// TIA Portal project "VGR_demo_rev2.0" (V16)

(* hardware
DEVICE "S7-1200 station_1"  S7-1200 Station
   slot 0: "Rack_0"  S7-1200 Rack  Rack  V1.0
   slot 1: "PLC_1"  CPU 1214C DC/DC/DC  6ES7 214-1AG40-0XB0  V4.4
   slot 2: "DI 16x24VDC/DQ 16xRelay_1"  6ES7 223-1BL32-0XB0  V2.0
   slot 3: "DI 16x24VDC/DQ 16xRelay_2"  6ES7 223-1BL32-0XB0  V2.0
*)

// ===== PLC "PLC_1"  CPU 1214C DC/DC/DC =====

VAR_GLOBAL   // PLC tag table "VGR - Vacuum Gripper Robot"
   "IX_VGR_RefSwitchVerticalAxis_I1" AT %I12.0 : Bool;   // VGR - I1 = Reference switch vertical axis
   "IX_VGR_RefSwitchHorizontalAxis_I2" AT %I12.1 : Bool;   // VGR - I2 = Reference switch horizontal axis
   "IX_VGR_RefSwitchRotate_I3" AT %I12.2 : Bool;   // VGR - I3 = Reference switch rotate
   "QX_VGR_M1_VerticalAxisUp_Q1" AT %Q13.0 : Bool;   // VGR - Q1 = Motor M1 vertical axis up
   "QX_VGR_M1_VerticalAxisDown_Q2" AT %Q13.1 : Bool;   // VGR - Q2 = Motor M1 vertical axis down
   "QX_VGR_M2_HorizontalAxisBackward_Q3" AT %Q13.2 : Bool;   // VGR - Q3 = Motor M2 horizontal axis backward
   "QX_VGR_M2_HorizontalAxisForward_Q4" AT %Q13.3 : Bool;   // VGR - Q4 = Motor M2 horizontal axis forward
   "QX_VGR_M3_RotateClockwise_Q5" AT %Q13.4 : Bool;   // VGR - Q5 = Motor M3 rotate clockwise
   "QX_VGR_M3_RotateCounterclockwise_Q6" AT %Q13.5 : Bool;   // VGR - Q6 = Motor M3 rotate counterclockwise
   "QX_VGR_Compressor_Q7" AT %Q13.6 : Bool;   // VGR - Q7 = Compressor
   "QX_VGR_ValveVacuum_Q8" AT %Q13.7 : Bool;   // VGR - Q8 = Valve vacuum
   "Enc_VGR_vertical" AT %ID1008 : DInt;
   "Enc_VGR_horizontal" AT %ID1012 : DInt;
   "Enc_VGR_rotate" AT %ID1016 : DInt;
END_VAR

VAR_GLOBAL   // PLC tag table "MPO - Multi Processing Station with Oven"
   "IX_MPO_RefSwitchOvenFeederInside_I6" AT %I8.5 : Bool;   // MPO - I6 = Reference switch oven feeder inside
   "IX_MPO_RefSwitchOvenFeederOutside_I7" AT %I8.6 : Bool;   // MPO - I7 = Reference switch oven feeder outside
   "QX_MPO_M4_OvenFeederRetract_Q5" AT %Q8.2 : Bool;   // MPO - Q5 = Motor M4 oven feeder retract
   "QX_MPO_M4_OvenFeederExtend_Q6" AT %Q8.3 : Bool;   // MPO - Q6 = Motor M4 oven feeder extend
   "QX_MPO_Compressor_Q10" AT %Q8.7 : Bool;   // MPO - Q10 = Compressor
   "QX_MPO_ValveOvenDoor_Q13" AT %Q9.2 : Bool;   // MPO - Q13 = Valve oven door
END_VAR

TYPE "typ_History"
   STRUCT
      ldt_ts : DTL;
      i_code : Int;
   END_STRUCT;
END_TYPE

TYPE "typ_Workpiece"
   STRUCT
      s_id : String;
      s_type : String;
      s_state : String;
   END_STRUCT;
END_TYPE

TYPE "typ_VGR"
   STRUCT
      x_Start_Park_Position : Bool;
      x_Park_Position_Reached : Bool;
      x_NFC_Start_First : Bool;
      x_NFC_Start : Bool;
      x_NFC_Completed : Bool;
      x_HBW_Storage : Bool;
      x_HBW_Outsource : Bool;
      s_HBW_Outsource_Typ : String;
      x_HBW_Discards : Bool;
      x_HBW_PickedUp : Bool;
      x_MPO_Req_Discard : Bool;
      x_MPO_Discards : Bool;
      x_Ready_For_Outsource : Bool;
      x_State_Process : Bool;
      x_Workpiece_NiO : Bool;
      horizontal_Axis : "typ_Axis";
      vertical_Axis : "typ_Axis";
      rotate_Axis : "typ_Axis";
      Workpiece : "typ_Workpiece";
      History : Array[1..20] of "typ_History";
      di_Pos_DSI_horizontal : DInt;
      di_Pos_DSI_Collect_vertical : DInt;
      di_Pos_DSI_Discard_vertical : DInt;
      di_Offset_Pos_DSI_NFC_vertical : DInt;
      di_Pos_DSI_rotate : DInt;
      di_Pos_DSO_horizontal : DInt;
      di_Pos_DSO_Collect_vertical : DInt;
      di_Pos_DSO_Discard_vertical : DInt;
      di_Offset_Pos_DSO_vertical : DInt;
      di_Pos_DSO_rotate : DInt;
      di_Pos_Color_horizontal : DInt;
      di_Pos_Color_vertical : DInt;
      di_Pos_Color_rotate : DInt;
      di_Pos_NFC_horizontal : DInt;
      di_Pos_NFC_vertical : DInt;
      di_Pos_NFC_rotate : DInt;
      di_Pos_MPO_horizontal : DInt;
      di_Pos_MPO_vertical : DInt;
      di_Offset_Pos_MPO_vertical : DInt;
      di_Pos_MPO_rotate : DInt;
      di_Pos_HBW_horizontal : DInt;
      di_Offset_Pos_HBW_horizontal : DInt;
      di_Pos_HBW_Collect_vertical : DInt;
      di_Pos_HBW_Discard_vertical : DInt;
      di_Offset_Pos_HBW_vertical : DInt;
      di_Pos_HBW_rotate : DInt;
      di_Pos_NiO_horizontal : DInt;
      di_Pos_NiO_vertical : DInt;
      di_Pos_NiO_rotate : DInt;
      di_Pos_SLD_Blue_horizontal : DInt;
      di_Pos_SLD_Blue_vertical : DInt;
      di_Pos_SLD_Blue_rotate : DInt;
      di_Pos_SLD_Red_horizontal : DInt;
      di_Pos_SLD_Red_vertical : DInt;
      di_Pos_SLD_Red_rotate : DInt;
      di_Pos_SLD_White_horizontal : DInt;
      di_Pos_SLD_White_vertical : DInt;
      di_Pos_SLD_White_rotate : DInt;
      di_Pos_Park_horizontal : DInt;
      di_Pos_Park_vertical : DInt;
      di_Pos_Park_rotate : DInt;
   END_STRUCT;
END_TYPE

TYPE "typ_SetupAxis"
   STRUCT
      x_Setup_Activ : Bool;   // Einrichten Kalibrieren aktiv / Set up calibration active
      i_AxisSelection : Int;   // Nummer der Achse / Number of the axis
      i_Function : Int;   // 0= Automatic, 10=Ref. Fahrt, 20= Tippen, 30=Tippen mit Schritweite, 40= Pos. Anfahren / 0 = automatic, 10 = ref. Travel, 20 = tap, 30 = tap with step width, 40 = start
      x_Set_Ref_Pos : Bool;   // Referenzwert setzen / Set reference value
      x_Set_Soft_End_Pos : Bool;   // Softwareendlagen setzen / Set software end positions
      x_Approach_Ref_Pos : Bool;   // Referenz anfahren / Approach reference
      x_Axis_Pos : Bool;   // Achse positiv / Axis positiv
      x_Axis_Neg : Bool;   // Achse negativ / Axis negative
      x_Approach_Target_Pos : Bool;   // Zielposition anfahren / Approach Target position
      w_Increment : Word;   // Inkremente pro Schritt / Increments per step
      i_PWM : Int;   // PWM Signal
      di_Target_Position : DInt;   // Zielposition / Target position
      di_ActualPosition : DInt;   // Aktuelle Position / Actual position
      di_Ref_Pos : DInt;   // Referenzposition / Reference position
      di_Actual_Ref_Pos : DInt;   // Aktuelle Referenzposition / Current reference position
      di_Soft_End_Pos_Neg : DInt;   // Softwareendlage negativ / Software end position negative
      di_Actual_Soft_End_Pos_Neg : DInt;   // Aktuelle Softwareendlage negativ / Current software end position negative
      di_Soft_End_Pos_Pos : DInt;   // Softwareendlage positiv / Software end position positiv
      di_Actual_Soft_End_Pos_Pos : DInt;   // Aktuelle Softwareendlage positiv / Current software end position positiv
      di_LoopValue : DInt;   // Schleifenwert / Loop value
   END_STRUCT;
END_TYPE

TYPE "typ_Axis_Data"
   STRUCT
      di_Pos_Soft_Switch : DInt := 0;
      di_Neg_Soft_Switch : DInt := 0;
      di_Ref_Pos : DInt := 0;
      di_Loop_Value : DInt := 0;
      di_Pos_Window : DInt := 15;
   END_STRUCT;
END_TYPE

TYPE "typ_Axis"
   STRUCT
      x_Start_Positioning : Bool;
      x_Reference : Bool;
      x_Referenced : Bool;
      x_Position_Reached : Bool;
      di_Target_Position : DInt;
      di_Increment : DInt;
      di_Actual_Position : DInt := 0;
      i_PWM : Int;
      Config : "typ_Axis_Data";
   END_STRUCT;
END_TYPE

TYPE "typ_Setup"
   STRUCT
      x_Clean_Rack_HBW : Bool;
      x_Park_Position : Bool;
      x_AcknowledgeButton : Bool;
      x_Color_Sensor_Calibration : Bool;
      x_Set_Calib_Value_Color_Blue : Bool;
      x_Set_Calib_Value_Color_White : Bool;
      x_Set_Calib_Value_Color_Red : Bool;
      x_Calculate_Value_Color : Bool;
      i_Color_Sensor_Selection : Int;
      w_Calib_ColorValue_Blue : Word;
      w_Calib_ColorValue_White : Word;
      w_Calib_ColorValue_Red : Word;
      w_Threshold_White_Red : Word;
      w_Threshold_Red_Blue : Word;
      w_Actual_ColorValue : Word;
      x_Set_Pos_Activ : Bool;   // Einrichten Kalibrieren aktiv / Set up calibration active
      x_Start_Positioning : Bool;
      x_Final_Positioning : Bool;
      x_Home_Positioning : Bool;
      x_Start_Offset : Bool;
      i_Pos_Selection : Int;   // Nummer der Achse / Number of the axis
      di_Pos_Horizontal : DInt;
      di_Pos_Vertical : DInt;
      di_Pos_Rotate : DInt;
      x_Counter_Value_Calibration : Bool;   // Einrichten Kalibrieren aktiv
      i_Calib_CounterValue_Blue : Int := 26;
      i_Calib_CounterValue_White : Int := 5;
      i_Calib_CounterValue_Red : Int := 16;
      x_Set_CounterValues : Bool;   // Einrichten Kalibrieren aktiv
      x_Activate_Continuous_Operation : Bool;
   END_STRUCT;
END_TYPE

// folder: 3.1. VGR

DATA_BLOCK "PRG_VGR_Demo_DB"   // DB1
{ S7_Optimized_Access := 'TRUE' }
VERSION : 0.1
// stored: InstanceOfName PRG_VGR_Demo
"PRG_VGR_Demo"
BEGIN
   di_Pos_Second_rotate := 885;
   di_Pos_Second_vertical_high := 450;
END_DATA_BLOCK

DATA_BLOCK "PRG_VGR_Axis_horizontal_DB"   // DB8
{ S7_Optimized_Access := 'TRUE' }
VERSION : 0.1
// stored: InstanceOfName PRG_VGR_Axis_horizontal
"PRG_VGR_Axis_horizontal"
BEGIN
END_DATA_BLOCK

DATA_BLOCK "PRG_VGR_Axis_vertical_DB"   // DB9
{ S7_Optimized_Access := 'TRUE' }
VERSION : 0.1
// stored: InstanceOfName PRG_VGR_Axis_vertical
"PRG_VGR_Axis_vertical"
BEGIN
END_DATA_BLOCK

DATA_BLOCK "PRG_VGR_Axis_rotate_DB"   // DB10
{ S7_Optimized_Access := 'TRUE' }
VERSION : 0.1
// stored: InstanceOfName PRG_VGR_Axis_rotate
"PRG_VGR_Axis_rotate"
BEGIN
END_DATA_BLOCK

DATA_BLOCK "PRG_VGR_Axis_horizontal_Act_Pos_DB"   // DB15
{ S7_Optimized_Access := 'TRUE' }
VERSION : 0.1
// stored: InstanceOfName PRG_VGR_Axis_horizontal_Act_Pos
"PRG_VGR_Axis_horizontal_Act_Pos"
BEGIN
END_DATA_BLOCK

DATA_BLOCK "PRG_VGR_Axis_vertical_Act_Pos_DB"   // DB29
{ S7_Optimized_Access := 'TRUE' }
VERSION : 0.1
// stored: InstanceOfName PRG_VGR_Axis_vertical_Act_Pos
"PRG_VGR_Axis_vertical_Act_Pos"
BEGIN
END_DATA_BLOCK

DATA_BLOCK "PRG_VGR_Axis_rotate_Act_Pos_DB"   // DB31
{ S7_Optimized_Access := 'TRUE' }
VERSION : 0.1
// stored: InstanceOfName PRG_VGR_Axis_rotate_Act_Pos
"PRG_VGR_Axis_rotate_Act_Pos"
BEGIN
END_DATA_BLOCK

// folder: 4. Global Declaration

DATA_BLOCK "gtyp_VGR"   // DB2
TITLE = Global DB VGR
{ S7_Optimized_Access := 'TRUE' }
AUTHOR : A.Schaefer
VERSION : 0.0
BEGIN
   di_Pos_DSI_Collect_vertical := 2950;
   di_Pos_MPO_vertical := 2000;
   di_Pos_HBW_Discard_vertical := 200;
   vertical_Axis.Config.di_Pos_Soft_Switch := 20000;
   horizontal_Axis.Config.di_Pos_Soft_Switch := 20000;
   rotate_Axis.Config.di_Pos_Soft_Switch := 20000;
   di_Pos_DSI_horizontal := 20;
   di_Pos_DSI_rotate := 30;
   di_Pos_Color_horizontal := 150;
   di_Pos_Color_rotate := 430;
   di_Pos_Color_vertical := 2450;
   di_Pos_NFC_vertical := 2450;
   di_Pos_NFC_horizontal := 900;
   di_Pos_NFC_rotate := 700;
   di_Pos_HBW_rotate := 5350;
   di_Offset_Pos_DSI_NFC_vertical := 1200;
   di_Offset_Pos_HBW_vertical := 100;
   di_Pos_HBW_horizontal := 600;
   di_Pos_SLD_Red_rotate := 1460;
   di_Pos_SLD_White_rotate := 1720;
   di_Pos_SLD_Blue_rotate := 1200;
   di_Pos_SLD_Red_vertical := 3100;
   di_Pos_SLD_White_vertical := 3100;
   di_Pos_SLD_Blue_vertical := 3100;
   di_Pos_SLD_Red_horizontal := 1580;
   di_Pos_SLD_White_horizontal := 1370;
   di_Pos_SLD_Blue_horizontal := 2150;
   di_Pos_DSO_rotate := 970;
   di_Pos_MPO_rotate := 3495;
   di_Pos_NiO_rotate := 1100;
   di_Pos_DSO_horizontal := 2070;
   di_Pos_DSO_Discard_vertical := 1480;
   di_Pos_NiO_vertical := 2700;
   di_Pos_MPO_horizontal := 3300;
   di_Pos_HBW_Collect_vertical := 650;
   di_Offset_Pos_MPO_vertical := 650;
   horizontal_Axis.i_PWM := 500;
   vertical_Axis.i_PWM := 800;
   rotate_Axis.i_PWM := 500;
   di_Offset_Pos_DSO_vertical := 500;
   di_Pos_Park_vertical := 3000;
   di_Pos_Park_rotate := 1750;
   di_Pos_Park_horizontal := 150;
   rotate_Axis.Config.di_Pos_Window := 15;
   vertical_Axis.Config.di_Pos_Window := 15;
   horizontal_Axis.Config.di_Pos_Window := 15;
END_DATA_BLOCK

DATA_BLOCK "gtyp_SetupAxis"   // DB4
TITLE = Global DB Setup Axis
{ S7_Optimized_Access := 'TRUE' }
AUTHOR : A.Schaefer
VERSION : 0.0
BEGIN
END_DATA_BLOCK

DATA_BLOCK "gtyp_Setup"   // DB23
TITLE = Global DB Setup
{ S7_Optimized_Access := 'TRUE' }
AUTHOR : A.Schaefer
VERSION : 0.0
BEGIN
END_DATA_BLOCK

// folder: (top level)

ORGANIZATION_BLOCK "Main"   // OB1, SCL, ProgramCycle
TITLE = "Main Program Sweep (Cycle)"
{ S7_Optimized_Access := 'TRUE' }
AUTHOR : A.Schaefer
VERSION : 0.0
BEGIN
   "PRG_VGR_Axis_horizontal_DB"();
   "PRG_VGR_Axis_vertical_DB"();
   "PRG_VGR_Axis_rotate_DB"();
   "PRG_VGR_Demo_DB"();
END_ORGANIZATION_BLOCK

ORGANIZATION_BLOCK "Cyclic interrupt"   // OB30, SCL, CyclicInterrupt
TITLE = Cyclic interrupt
{ S7_Optimized_Access := 'TRUE' }
AUTHOR : A.Schaefer
VERSION : 0.0
   VAR_TEMP
      li_Return_LDT : Int;
   END_VAR
BEGIN
   "PRG_VGR_Axis_horizontal_Act_Pos_DB"();
   "PRG_VGR_Axis_vertical_Act_Pos_DB"();
   "PRG_VGR_Axis_rotate_Act_Pos_DB"();
END_ORGANIZATION_BLOCK

ORGANIZATION_BLOCK "Startup"   // OB100, SCL, Startup
TITLE = "Complete Restart"
{ S7_Optimized_Access := 'TRUE' }
VERSION : 0.1
   VAR_INPUT
      LostRetentive : Bool;   // True if retentive data are lost
      LostRTC : Bool;   // True if date and time are lost
   END_VAR
BEGIN
   "PRG_VGR_Demo_DB".li_StepCase := 0;
END_ORGANIZATION_BLOCK

// folder: 1. FB / FC

FUNCTION_BLOCK "FB_INC_DEC"   // FB9, SCL
TITLE = Funktionblock Increment decodition
{ S7_Optimized_Access := 'TRUE' }
AUTHOR : A.Schaefer
VERSION : 0.0
   VAR_INPUT
      inx_CHa : Bool := false;
      inx_CHb : Bool := false;
      inx_RST : Bool := False;
      ini_Ref_Wert : Int := 0;
   END_VAR
   VAR_OUTPUT
      outx_dir : Bool := false;
      outi_cnt : Int := 0;
   END_VAR
   VAR
      lx_edgea : Bool := False;
      lx_clka : Bool;
      lx_clkb : Bool;
      lx_edgeb : Bool;
      lx_axb : Bool;
      lx_dir : Bool;
      li_cnt : Int;
   END_VAR
BEGIN

   #lx_axb := #inx_CHa XOR #inx_CHb;

   (* create pulses for channel a *)
   #lx_clka := #inx_CHa XOR #lx_edgea;
   #lx_edgea := #inx_CHa;

   #lx_clkb := #inx_CHb XOR #lx_edgeb;
   #lx_edgeb := #inx_CHb;

   (* create pulses for both channels *)
   #lx_clka := #lx_clka OR #lx_clkb;

   (* set the direction output *)
   IF #lx_axb AND #lx_clka THEN
       #lx_dir := TRUE;
   END_IF;
   IF #lx_axb AND #lx_clkb THEN
       #lx_dir := FALSE;
   END_IF;

   (* increment or decrement the counter *)
   IF #lx_clka AND #lx_dir THEN
       #li_cnt := #li_cnt + 1;
   END_IF;
   IF #lx_clka AND NOT #lx_dir THEN
       #li_cnt := #li_cnt - 1;
   END_IF;

   (* reset the counter if rst active *)
   IF #inx_RST THEN
       #li_cnt := #ini_Ref_Wert;
   END_IF;

   #outx_dir := #lx_dir;
   #outi_cnt := #li_cnt;
END_FUNCTION_BLOCK

FUNCTION_BLOCK "FB_Axis"   // FB22, SCL
TITLE = Functionblock Axis
{ S7_Optimized_Access := 'TRUE' }
AUTHOR : A.Schaefer
VERSION : 0.0
   VAR_INPUT
      ini_Axis : Int;
      indi_Increment : DInt;
      inx_Ref_Switch : Bool;
      inx_Start_Positioning : Bool;
      inx_Referencing : Bool;
      ini_PWM : Int;
      indi_Target_Position : DInt;
   END_VAR
   VAR_OUTPUT
      outx_Referenced : Bool;
      outx_Position_Reached : Bool;
      outx_Motor_Pos : Bool;
      outx_Motor_Neg : Bool;
      outi_Motor_PWM : Int;
      outdi_Actual_Position : DInt;
   END_VAR
   VAR_IN_OUT
      inouttyp_Config : "typ_Axis_Data";
      inouttyp_Setup : "typ_SetupAxis";
   END_VAR
   VAR
      li_StepCaseSetup : Int;
      li_StepCase : Int;
      lx_Init : Bool;
      lx_Motor_Neg : Bool;
      lx_Motor_Pos : Bool;
      lx_Start_TON_Wait : Bool;
      li_PWM : Int;
      ldi_ValueStep : DInt;
      ldi_Actual_Position : DInt;
      ldi_Actual_Position_Old : DInt;
      lfb_R_Trig_Setup : R_TRIG;
      lfb_R_Trig_Referencing : R_TRIG;
      lfb_TON_Wait : TON_TIME;
   END_VAR
BEGIN
   IF #lx_Init THEN

       // rising edge set up axis
       #lfb_R_Trig_Setup(CLK := #inouttyp_Setup.x_Setup_Activ);

       //Reload when switching to set up
       IF #lfb_R_Trig_Setup.Q THEN
           #inouttyp_Setup.di_LoopValue               := #inouttyp_Config.di_Loop_Value;
           #inouttyp_Setup.di_Ref_Pos                 := 
           #inouttyp_Setup.di_Actual_Ref_Pos          := #inouttyp_Config.di_Ref_Pos;
           #inouttyp_Setup.di_Soft_End_Pos_Neg        := 
           #inouttyp_Setup.di_Actual_Soft_End_Pos_Neg := #inouttyp_Config.di_Neg_Soft_Switch;
           #inouttyp_Setup.di_Soft_End_Pos_Pos        :=
           #inouttyp_Setup.di_Actual_Soft_End_Pos_Pos := #inouttyp_Config.di_Pos_Soft_Switch;
           #inouttyp_Setup.i_PWM                      := #ini_PWM;
           #inouttyp_Setup.x_Approach_Ref_Pos         := FALSE;
           #inouttyp_Setup.x_Approach_Target_Pos      := FALSE;
           #inouttyp_Setup.x_Axis_Neg                 := FALSE;
           #inouttyp_Setup.x_Axis_Pos                 := FALSE;
           #inouttyp_Setup.x_Set_Ref_Pos              := FALSE;
           #inouttyp_Setup.x_Set_Soft_End_Pos         := FALSE;
       END_IF;

       #ldi_Actual_Position := #indi_Increment;

       //rising edge referencing
       #lfb_R_Trig_Referencing(CLK := #inx_Referencing);

       //waiting period
       #lfb_TON_Wait(IN := #lx_Start_TON_Wait,
                     PT := T#200ms);

       (**********************************)
       (******   set up step chain   *****)
       (**********************************)
       IF #inouttyp_Setup.i_AxisSelection = #ini_Axis AND #inouttyp_Setup.x_Setup_Activ THEN
           IF #inouttyp_Setup.x_Approach_Ref_Pos THEN
               #inouttyp_Setup.i_Function := 10;
           END_IF;

           CASE #inouttyp_Setup.i_Function OF

               0:  // automatic
                   #ldi_Actual_Position_Old := 0;
                   #inouttyp_Setup.x_Approach_Ref_Pos := FALSE;
                   #lx_Start_TON_Wait := FALSE;

               10: // homing
                   IF #inouttyp_Setup.x_Approach_Ref_Pos THEN
                       IF NOT #inx_Ref_Switch THEN
                           #lx_Motor_Neg := TRUE;
                           #lx_Motor_Pos := FALSE;
                           #outx_Referenced := FALSE;
                       END_IF;

                       IF #inx_Ref_Switch THEN
                           #lx_Motor_Neg := TRUE;
                           #lx_Motor_Pos := TRUE;

                           IF #ldi_Actual_Position = #inouttyp_Config.di_Ref_Pos THEN
                               #inouttyp_Setup.x_Approach_Ref_Pos := FALSE;
                               #lx_Motor_Neg       := FALSE;
                               #lx_Motor_Pos       := FALSE;
                               #outx_Referenced    := TRUE;
                           END_IF;
                       END_IF;
                   END_IF;

               20:  // tap
                   #lx_Motor_Neg := #inouttyp_Setup.x_Axis_Neg AND NOT #inx_Ref_Switch AND NOT (#ldi_Actual_Position <= #inouttyp_Setup.di_Soft_End_Pos_Neg);
                   #lx_Motor_Pos := #inouttyp_Setup.x_Axis_Pos AND NOT #lx_Motor_Neg AND NOT (#ldi_Actual_Position >= #inouttyp_Setup.di_Soft_End_Pos_Pos);

               30:  // tap with increment
                   #ldi_Actual_Position_Old := #ldi_Actual_Position;

                   // positiv
                   IF #inouttyp_Setup.x_Axis_Pos AND NOT ((#ldi_Actual_Position + #inouttyp_Setup.w_Increment + #inouttyp_Setup.di_LoopValue) >= #inouttyp_Setup.di_Soft_End_Pos_Pos) THEN
                       #lx_Motor_Neg := FALSE;
                       #lx_Motor_Pos := TRUE;
                       #ldi_ValueStep := #ldi_Actual_Position_Old + #inouttyp_Setup.w_Increment;

                       // without loop
                       IF (#inouttyp_Setup.di_LoopValue = 0) THEN
                           #inouttyp_Setup.i_Function := 36;
                       ELSE
                           #inouttyp_Setup.i_Function := 31;
                       END_IF;
                   // negativ
                   ELSIF #inouttyp_Setup.x_Axis_Neg AND NOT ((#ldi_Actual_Position - #inouttyp_Setup.w_Increment) <= #inouttyp_Config.di_Neg_Soft_Switch) THEN
                       #lx_Motor_Neg := TRUE;
                       #lx_Motor_Pos := FALSE;
                       #ldi_ValueStep := #ldi_Actual_Position_Old - #inouttyp_Setup.w_Increment;
                       #inouttyp_Setup.i_Function := 34;
                   END_IF;

               31: // with loop
                   IF ((#ldi_Actual_Position >= (#ldi_ValueStep + #inouttyp_Setup.di_LoopValue - #inouttyp_Config.di_Pos_Window)) = 0) THEN
                       #lx_Motor_Neg := TRUE;
                       #lx_Motor_Pos := TRUE;
                       #inouttyp_Setup.i_Function := 32;
                   END_IF;

               32: // wait sequence
                   #lx_Start_TON_Wait := TRUE;

                   IF #lfb_TON_Wait.Q THEN
                       #lx_Motor_Neg               := FALSE;
                       #lx_Motor_Pos               := FALSE;
                       #lx_Start_TON_Wait          := FALSE;
                       #inouttyp_Setup.i_Function  := 33;
                   END_IF;

               33: // change direction
                   #lx_Motor_Neg := TRUE;
                   #lx_Motor_Pos := FALSE;
                   #inouttyp_Setup.i_Function := 34;

               34: // position reached negativ
                   IF (#ldi_Actual_Position <= (#ldi_ValueStep + #inouttyp_Config.di_Pos_Window))
                       AND (#ldi_Actual_Position >= (#ldi_ValueStep - #inouttyp_Config.di_Pos_Window)) THEN
                       #lx_Motor_Neg := TRUE;
                       #lx_Motor_Pos := TRUE;
                       #inouttyp_Setup.i_Function := 35;
                   END_IF;

               35: // wait sequence
                   #lx_Start_TON_Wait := TRUE;

                   IF #lfb_TON_Wait.Q THEN
                       #lx_Motor_Neg := FALSE;
                       #lx_Motor_Pos := FALSE;
                       #lx_Start_TON_Wait := FALSE;
                       #inouttyp_Setup.x_Axis_Neg := FALSE;
                       #inouttyp_Setup.x_Axis_Pos := FALSE;
                       #inouttyp_Setup.i_Function := 30;
                   END_IF;


               36: // position reached positiv
                   IF (#ldi_Actual_Position <= (#ldi_ValueStep + #inouttyp_Config.di_Pos_Window))
                       AND (#ldi_Actual_Position >= (#ldi_ValueStep - #inouttyp_Config.di_Pos_Window)) THEN
                       #lx_Motor_Neg := TRUE;
                       #lx_Motor_Pos := TRUE;
                       #inouttyp_Setup.i_Function := 37;
                   END_IF;

               37: // wait sequence
                   #lx_Start_TON_Wait := TRUE;

                   IF #lfb_TON_Wait.Q THEN
                       #lx_Motor_Neg := FALSE;
                       #lx_Motor_Pos := FALSE;
                       #lx_Start_TON_Wait := FALSE;
                       #inouttyp_Setup.x_Axis_Neg := FALSE;
                       #inouttyp_Setup.x_Axis_Pos := FALSE;
                       #inouttyp_Setup.i_Function := 30;
                   END_IF;

               40: // approach position
                   IF #inouttyp_Setup.x_Approach_Target_Pos THEN
                       // positiv
                       IF (#inouttyp_Setup.di_Target_Position > #ldi_Actual_Position) AND NOT ((#inouttyp_Setup.di_Target_Position + #inouttyp_Setup.di_LoopValue) >= #inouttyp_Setup.di_Soft_End_Pos_Pos)  THEN
                           #lx_Motor_Neg := FALSE;
                           #lx_Motor_Pos := TRUE;
                           // without loop
                           IF (#inouttyp_Setup.di_LoopValue = 0) THEN
                               #inouttyp_Setup.i_Function := 46;
                           ELSE
                               #inouttyp_Setup.i_Function := 41;
                           END_IF;
                       // negativ
                       ELSIF ((#inouttyp_Setup.di_Target_Position < #ldi_Actual_Position) AND NOT (#inouttyp_Setup.di_Target_Position <= #inouttyp_Config.di_Neg_Soft_Switch))  THEN
                           #lx_Motor_Neg := TRUE;
                           #lx_Motor_Pos := FALSE;
                           #inouttyp_Setup.i_Function := 44;
                       ELSIF (#inouttyp_Setup.di_Target_Position = #ldi_Actual_Position) THEN
                           #inouttyp_Setup.i_Function := 46;
                       END_IF;

                   END_IF;

               41: // with loop
                   IF (#ldi_Actual_Position >= (#inouttyp_Setup.di_Target_Position + #inouttyp_Setup.di_LoopValue - #inouttyp_Config.di_Pos_Window)) THEN
                       #lx_Motor_Neg := TRUE;
                       #lx_Motor_Pos := TRUE;
                       #inouttyp_Setup.i_Function := 42;
                   END_IF;

               42: // wait sequence
                   #lx_Start_TON_Wait := TRUE;

                   IF #lfb_TON_Wait.Q THEN
                       #lx_Motor_Neg := FALSE;
                       #lx_Motor_Pos := FALSE;
                       #lx_Start_TON_Wait := FALSE;
                       #inouttyp_Setup.i_Function := 43;
                   END_IF;

               43: // change direction
                   #lx_Motor_Neg   := TRUE;
                   #lx_Motor_Pos   := FALSE;
                   #inouttyp_Setup.i_Function     := 44;

               44: // position reached negativ
                   IF (#ldi_Actual_Position <= (#inouttyp_Setup.di_Target_Position + #inouttyp_Config.di_Pos_Window))
                       AND (#ldi_Actual_Position >= (#inouttyp_Setup.di_Target_Position - #inouttyp_Config.di_Pos_Window)) THEN
                       #lx_Motor_Neg := TRUE;
                       #lx_Motor_Pos := TRUE;
                       #inouttyp_Setup.i_Function := 45;
                   END_IF;

               45: // wait sequence
                   #lx_Start_TON_Wait := TRUE;

                   IF #lfb_TON_Wait.Q THEN
                       #lx_Motor_Neg := FALSE;
                       #lx_Motor_Pos := FALSE;
                       #lx_Start_TON_Wait := FALSE;
                       #inouttyp_Setup.x_Axis_Neg := FALSE;
                       #inouttyp_Setup.x_Axis_Pos := FALSE;
                       #inouttyp_Setup.i_Function := 40;
                   END_IF;

               46: //  position reached positiv
                   IF (#ldi_Actual_Position <= (#inouttyp_Setup.di_Target_Position + #inouttyp_Config.di_Pos_Window))
                       AND (#ldi_Actual_Position >= (#inouttyp_Setup.di_Target_Position - #inouttyp_Config.di_Pos_Window)) THEN
                       #lx_Motor_Neg := TRUE;
                       #lx_Motor_Pos := TRUE;
                       #inouttyp_Setup.i_Function := 47;
                   END_IF;

               47:  // wait sequence
                   #lx_Start_TON_Wait := TRUE;

                   IF #lfb_TON_Wait.Q THEN
                       #lx_Motor_Neg := FALSE;
                       #lx_Motor_Pos := FALSE;
                       #lx_Start_TON_Wait := FALSE;
                       #inouttyp_Setup.x_Approach_Target_Pos := FALSE;
                       #inouttyp_Setup.i_Function := 40;
                   END_IF;
               ELSE  // Statement section ELSE
                   ;
           END_CASE;

           // set reference point
           IF #inouttyp_Setup.x_Set_Ref_Pos THEN
               #inouttyp_Setup.di_Actual_Ref_Pos   :=
               #inouttyp_Config.di_Ref_Pos         := #inouttyp_Setup.di_Ref_Pos;
               #inouttyp_Setup.x_Set_Ref_Pos       := FALSE;
           END_IF;

           // set software end position
           IF #inouttyp_Setup.x_Set_Soft_End_Pos THEN
               #inouttyp_Setup.di_Actual_Soft_End_Pos_Neg  :=
               #inouttyp_Config.di_Neg_Soft_Switch         := #inouttyp_Setup.di_Soft_End_Pos_Neg;
               #inouttyp_Setup.di_Actual_Soft_End_Pos_Pos  :=
               #inouttyp_Config.di_Pos_Soft_Switch         := #inouttyp_Setup.di_Soft_End_Pos_Pos;
               #inouttyp_Setup.x_Set_Soft_End_Pos := FALSE;
           END_IF;

           // reload PWM
           #li_PWM := #inouttyp_Setup.i_PWM;

           // reload actual position
           #inouttyp_Setup.di_ActualPosition           := #ldi_Actual_Position;

       (************************************)
       (******   position step chain   *****)
       (************************************)
       ELSIF NOT #inouttyp_Setup.x_Setup_Activ THEN

           // rising edge set up axis
           IF #lfb_R_Trig_Referencing.Q THEN
               #li_StepCase := 0;
           END_IF;

           CASE #li_StepCase OF

               0:  // init
                   #lx_Start_TON_Wait := FALSE;

                   IF #inx_Referencing THEN
                       #li_StepCase            := 10;
                       #outx_Position_Reached  := FALSE;
                       #outx_Referenced        := FALSE;
                   ELSIF #inx_Start_Positioning THEN
                       #li_StepCase            := 20;
                       #outx_Position_Reached  := FALSE;
                   END_IF;

               10: // homing
                   IF NOT #inx_Ref_Switch THEN
                       #lx_Motor_Neg := TRUE;
                       #lx_Motor_Pos := FALSE;
                   END_IF;

                   IF #inx_Ref_Switch THEN
                       #lx_Motor_Neg := TRUE;
                       #lx_Motor_Pos := TRUE;

                       IF #inx_Ref_Switch THEN
                           IF #ldi_Actual_Position = #inouttyp_Config.di_Ref_Pos THEN
                               #lx_Motor_Neg := FALSE;
                               #lx_Motor_Pos := FALSE;
                               #outx_Referenced := TRUE;
                               #li_StepCase := 11;
                           END_IF;
                       END_IF;
                   END_IF;

               11: // wait not referencing
                   IF NOT #inx_Referencing THEN
                       #li_StepCase := 0;
                   END_IF;

               20: // approach position
                   // positiv
                   IF (#indi_Target_Position > #ldi_Actual_Position) AND NOT ((#indi_Target_Position + #inouttyp_Config.di_Loop_Value) >= #inouttyp_Config.di_Pos_Soft_Switch) THEN
                       #lx_Motor_Neg := FALSE;
                       #lx_Motor_Pos := TRUE;
                       //without loop
                       IF (#inouttyp_Config.di_Loop_Value = 0) THEN
                           #li_StepCase := 26;
                       ELSE
                           #li_StepCase := 21;
                       END_IF;
                   // negativ
                   ELSIF ((#indi_Target_Position < #ldi_Actual_Position) AND NOT (#indi_Target_Position <= #inouttyp_Config.di_Neg_Soft_Switch)) THEN
                       #lx_Motor_Neg := TRUE;
                       #lx_Motor_Pos := FALSE;
                       #li_StepCase := 24;
                   ELSIF (#indi_Target_Position = #ldi_Actual_Position) THEN
                       #li_StepCase := 26;
                   END_IF;

               21: // with loop
                   IF (#ldi_Actual_Position >= (#indi_Target_Position + #inouttyp_Config.di_Loop_Value - #inouttyp_Config.di_Pos_Window)) THEN
                       #lx_Motor_Neg := TRUE;
                       #lx_Motor_Pos := TRUE;
                       #li_StepCase := 22;
                   END_IF;

               22: // wait sequence
                   #lx_Start_TON_Wait := TRUE;

                   IF #lfb_TON_Wait.Q THEN
                       #lx_Motor_Neg := FALSE;
                       #lx_Motor_Pos := FALSE;
                       #lx_Start_TON_Wait := FALSE;
                       #inouttyp_Setup.i_Function := 23;
                   END_IF;

               23: // change direction
                   #lx_Motor_Neg := TRUE;
                   #lx_Motor_Pos := FALSE;
                   #li_StepCase := 24;

               24: // position reached negativ
                   IF (#ldi_Actual_Position <= (#indi_Target_Position + #inouttyp_Config.di_Pos_Window))
                       AND (#ldi_Actual_Position >= (#indi_Target_Position - #inouttyp_Config.di_Pos_Window)) THEN
                       #lx_Motor_Neg := TRUE;
                       #lx_Motor_Pos := TRUE;
                       #li_StepCase := 25;
                   END_IF;

               25: // wait sequence
                   #lx_Start_TON_Wait := TRUE;

                   IF #lfb_TON_Wait.Q THEN
                       #lx_Motor_Neg := FALSE;
                       #lx_Motor_Pos := FALSE;
                       #lx_Start_TON_Wait := FALSE;
                       #outx_Position_Reached := TRUE;
                       #li_StepCase := 28;
                   END_IF;

               26: // position reached positiv
                   IF (#ldi_Actual_Position <= (#indi_Target_Position + #inouttyp_Config.di_Pos_Window))
                       AND (#ldi_Actual_Position >= (#indi_Target_Position - #inouttyp_Config.di_Pos_Window)) THEN
                       #lx_Motor_Neg := TRUE;
                       #lx_Motor_Pos := TRUE;
                       #li_StepCase := 27;
                   END_IF;

               27: // wait sequence
                   #lx_Start_TON_Wait := TRUE;

                   IF #lfb_TON_Wait.Q THEN
                       #lx_Motor_Neg := FALSE;
                       #lx_Motor_Pos := FALSE;
                       #lx_Start_TON_Wait := FALSE;
                       #outx_Position_Reached := TRUE;
                       #li_StepCase := 28;
                   END_IF;

               28: // wait not start positioning
                   IF NOT #inx_Start_Positioning THEN
                       #li_StepCase := 0;
                   END_IF;
               // statement section ELSE    
               ELSE  
                   ;
           END_CASE;

           // reload PWM
           #li_PWM := #ini_PWM;
       END_IF;

       // reload outputs
       #outx_Motor_Neg         := #lx_Motor_Neg;
       #outx_Motor_Pos         := #lx_Motor_Pos;
       #outi_Motor_PWM         := #li_PWM;
       #outdi_Actual_Position  := #ldi_Actual_Position;

   ELSE
       #lx_Init := TRUE;
   END_IF;
END_FUNCTION_BLOCK

FUNCTION "FC_Scale_linear" : Real   // FC1, SCL
TITLE = Function scale linear
{ S7_Optimized_Access := 'TRUE' }
AUTHOR : A.Schaefer
VERSION : 0.0
   VAR_INPUT
      inr_Y1 : Real;   // Skalierungs-Anfangswert für Y (OUTPUT) / Initial scaling value for Y (INPUT)
      inr_Y2 : Real;   // Skalierungs-Endwert für Y (OUTPUT) / Scaling end value for Y (INPUT)
      inr_X1 : Real;   // Skalierungs-Anfangswert für X (INPUT) / Initial scaling value for X (INPUT)
      inr_X2 : Real;   // Skalierungs-Endwert für X (INPUT) / Scaling end value for X (INPUT)
      inr_X : Real;   // Zu Skalierender Wert / Value to be scaled
   END_VAR
   VAR_TEMP
      lr_y_delta : Real;   // Temp delta y
      lr_x_delta : Real;   // Temp delta x
      lr_m : Real;   // Temp gradient m
   END_VAR
   // Ret_Val : Return result
BEGIN
   (********************************************************)
   (* FC for linear scaling. Line function  y=m*(x-x1)+y1  *)
   (********************************************************)

   #lr_y_delta := (#inr_Y2 - #inr_Y1);
   #lr_x_delta := (#inr_X2 - #inr_X1);

   IF #lr_y_delta <> 0 AND #lr_x_delta <> 0 THEN
       #lr_m := (#lr_y_delta / #lr_x_delta);
       #FC_Scale_linear := (#lr_m * (#inr_X - #inr_X1)) + #inr_Y1;
   ELSE
       #FC_Scale_linear := 0;
   END_IF;
END_FUNCTION

// folder: 3.1. VGR

FUNCTION_BLOCK "PRG_VGR_Axis_vertical"   // FB1, SCL
TITLE = Program Axis vertical VGR
{ S7_Optimized_Access := 'TRUE' }
AUTHOR : A.Schaefer
VERSION : 0.0
   VAR
      lx_Init : Bool;
      lfb_vertical_Axis : "FB_Axis";
   END_VAR
BEGIN
   IF #lx_Init THEN

       // FB Axis vertical
       #lfb_vertical_Axis(ini_Axis         := 2,
                   indi_Increment          := "gtyp_VGR".vertical_Axis.di_Increment,
                   inx_Ref_Switch          := "IX_VGR_RefSwitchVerticalAxis_I1",
                   inx_Referencing         := "gtyp_VGR".vertical_Axis.x_Reference,
                   inx_Start_Positioning   := "gtyp_VGR".vertical_Axis.x_Start_Positioning,
                   indi_Target_Position    := "gtyp_VGR".vertical_Axis.di_Target_Position,
                   ini_PWM                 := "gtyp_VGR".vertical_Axis.i_PWM,
                   inouttyp_Config         := "gtyp_VGR".vertical_Axis.Config,
                   inouttyp_Setup          := "gtyp_SetupAxis");

       "QX_VGR_M1_VerticalAxisUp_Q1"       := #lfb_vertical_Axis.outx_Motor_Neg;
       "QX_VGR_M1_VerticalAxisDown_Q2"     := #lfb_vertical_Axis.outx_Motor_Pos;
       "gtyp_VGR".vertical_Axis.di_Actual_Position:= #lfb_vertical_Axis.outdi_Actual_Position;
       "gtyp_VGR".vertical_Axis.x_Referenced      := #lfb_vertical_Axis.outx_Referenced;
       "gtyp_VGR".vertical_Axis.x_Position_Reached:= #lfb_vertical_Axis.outx_Position_Reached;
   ELSE
       #lx_Init := TRUE;
   END_IF;
END_FUNCTION_BLOCK

FUNCTION_BLOCK "PRG_VGR_Demo"   // FB3, SCL
{ S7_Optimized_Access := 'TRUE' }
VERSION : 0.1
   VAR
      li_StepCase : Int;
      lx_Start_TON_Wait : Bool;
      lx_Start_TON_State : Bool;
      lt_TON_Wait : Time;
      lx_Init : Bool := true;
      di_Pos_First_rotate : DInt := 1770;
      di_Pos_First_horizontal : DInt := 1370;
      di_Pos_First_vertical : DInt := 3100;
      di_Pos_Second_vertical_high : DInt := 350;
      di_Pos_Second_rotate : DInt := 400;
      di_Pos_Second_horizontal : DInt := 850;
      di_Pos_Second_vertical : DInt := 500;
      lfb_TON_Wait : TON_TIME;
   END_VAR
BEGIN
   IF #lx_Init THEN

       // FB TON Wait
       #lfb_TON_Wait(IN := #lx_Start_TON_Wait,
                     PT := #lt_TON_Wait);

       // конечный автомат VGR
       CASE #li_StepCase OF

           0: // инициализация
               #lx_Start_TON_Wait := FALSE;
               "gtyp_VGR".horizontal_Axis.x_Start_Positioning := FALSE;
               "gtyp_VGR".vertical_Axis.x_Start_Positioning := FALSE;
               "gtyp_VGR".rotate_Axis.x_Start_Positioning := FALSE;
               "gtyp_VGR".x_Ready_For_Outsource := FALSE;
               "QX_VGR_Compressor_Q7" := FALSE;
               "QX_VGR_ValveVacuum_Q8" := FALSE;
               #li_StepCase := 10;

           10: // парковка вертикальной оси
               "gtyp_VGR".vertical_Axis.x_Reference := TRUE;

               IF NOT "gtyp_VGR".vertical_Axis.x_Referenced THEN
                   #li_StepCase := 20;
               END_IF;

           20: // завершение парковки вертикальной оси
               IF "gtyp_VGR".vertical_Axis.x_Referenced THEN
                   "gtyp_VGR".vertical_Axis.x_Reference := FALSE;
                   #li_StepCase := 30;
               END_IF;

           30: // парковка горизонтальной оси
               "gtyp_VGR".horizontal_Axis.x_Reference := TRUE;

               IF NOT "gtyp_VGR".horizontal_Axis.x_Referenced THEN
                   #li_StepCase := 40;
               END_IF;

           40: // завершение парковки горизонтальной оси
               IF "gtyp_VGR".horizontal_Axis.x_Referenced THEN
                   "gtyp_VGR".horizontal_Axis.x_Reference := FALSE;
                   #li_StepCase := 50;
               END_IF;

           50: // парковка платформы
               "gtyp_VGR".rotate_Axis.x_Reference := TRUE;

               IF NOT "gtyp_VGR".rotate_Axis.x_Referenced THEN
                   #li_StepCase := 60;
               END_IF;

           60: // завершение парковки платформы
               IF "gtyp_VGR".rotate_Axis.x_Referenced THEN
                   "gtyp_VGR".rotate_Axis.x_Reference := FALSE;

                   // если механизм загрузки в печь не в позиции снаружи - выдвинуть механизм загрузки
                   IF NOT "IX_MPO_RefSwitchOvenFeederOutside_I7" THEN
                       #li_StepCase := 61;
                   ELSE
                       #li_StepCase := 70;
                   END_IF;
               END_IF;

            61: // включить компрессор MPO
                "QX_MPO_Compressor_Q10" := TRUE;

                #lx_Start_TON_Wait := TRUE;
                #lt_TON_Wait := T#1000ms;

                IF #lfb_TON_Wait.Q THEN
                    #lx_Start_TON_Wait := FALSE;
                    #li_StepCase := 62;
                END_IF;

            62: // открыть дверь MPO
                "QX_MPO_ValveOvenDoor_Q13" := TRUE;

                #lx_Start_TON_Wait := TRUE;
                #lt_TON_Wait := T#2000ms;

                IF #lfb_TON_Wait.Q THEN
                    #lx_Start_TON_Wait := FALSE;
                    #li_StepCase := 63;
                END_IF;

            63: // выдвинуть механизм загрузки. Если выдвинут - опустить дверь и выключить компрессор.
                "QX_MPO_M4_OvenFeederRetract_Q5" := FALSE;
                "QX_MPO_M4_OvenFeederExtend_Q6" := TRUE;

                IF "IX_MPO_RefSwitchOvenFeederOutside_I7" AND NOT "IX_MPO_RefSwitchOvenFeederInside_I6" THEN
                    "QX_MPO_M4_OvenFeederRetract_Q5" := FALSE;
                    "QX_MPO_M4_OvenFeederExtend_Q6" := FALSE;
                    "QX_MPO_ValveOvenDoor_Q13" := FALSE;
                    "QX_MPO_Compressor_Q10" := FALSE;
                    #li_StepCase := 70;
                END_IF;

           (*************************************************)
           (****  Взять деталь из кармана белых деталей  ****)
           (*************************************************)     

           70:   // вращение платформы
               "gtyp_VGR".rotate_Axis.di_Target_Position := "gtyp_VGR".di_Pos_SLD_White_rotate;
               "gtyp_VGR".rotate_Axis.x_Start_Positioning := TRUE;

               IF ("gtyp_VGR".rotate_Axis.di_Actual_Position <= ("gtyp_VGR".di_Pos_SLD_White_rotate + "gtyp_VGR".rotate_Axis.Config.di_Pos_Window))
                   AND ("gtyp_VGR".rotate_Axis.di_Actual_Position >= ("gtyp_VGR".di_Pos_SLD_White_rotate - "gtyp_VGR".rotate_Axis.Config.di_Pos_Window))
                   AND "gtyp_VGR".rotate_Axis.x_Position_Reached THEN
                   "gtyp_VGR".rotate_Axis.x_Start_Positioning := FALSE;
                   #li_StepCase := 80;
               END_IF;

           80:   // горизонтальная ось вперед
               "gtyp_VGR".horizontal_Axis.di_Target_Position := "gtyp_VGR".di_Pos_SLD_White_horizontal;
               "gtyp_VGR".horizontal_Axis.x_Start_Positioning := TRUE;

               IF ("gtyp_VGR".horizontal_Axis.di_Actual_Position <= ("gtyp_VGR".di_Pos_SLD_White_horizontal + "gtyp_VGR".horizontal_Axis.Config.di_Pos_Window))
                   AND ("gtyp_VGR".horizontal_Axis.di_Actual_Position >= ("gtyp_VGR".di_Pos_SLD_White_horizontal - "gtyp_VGR".horizontal_Axis.Config.di_Pos_Window))
                   AND "gtyp_VGR".horizontal_Axis.x_Position_Reached THEN
                   "gtyp_VGR".horizontal_Axis.x_Start_Positioning := FALSE;
                   #li_StepCase := 90;
               END_IF;

            90:    // вертикальная ось вниз
                "gtyp_VGR".vertical_Axis.di_Target_Position := "gtyp_VGR".di_Pos_SLD_White_vertical;
                "gtyp_VGR".vertical_Axis.x_Start_Positioning := TRUE;

                IF ("gtyp_VGR".vertical_Axis.di_Actual_Position <= ("gtyp_VGR".di_Pos_SLD_White_vertical + "gtyp_VGR".vertical_Axis.Config.di_Pos_Window))
                    AND ("gtyp_VGR".vertical_Axis.di_Actual_Position >= ("gtyp_VGR".di_Pos_SLD_White_vertical - "gtyp_VGR".vertical_Axis.Config.di_Pos_Window))
                    AND "gtyp_VGR".vertical_Axis.x_Position_Reached THEN
                    "gtyp_VGR".vertical_Axis.x_Start_Positioning := FALSE;
                    #li_StepCase := 100;
                END_IF;

            100:    // запуск компрессора
                "QX_VGR_Compressor_Q7" := TRUE;

                #lx_Start_TON_Wait := TRUE;
                #lt_TON_Wait := T#1000ms;

                IF #lfb_TON_Wait.Q THEN
                    #lx_Start_TON_Wait := FALSE;
                    #li_StepCase := 110;
                END_IF;

            110:    // включение клапана (захват детали)
                "QX_VGR_ValveVacuum_Q8" := true;

                #lx_Start_TON_Wait := TRUE;
                #lt_TON_Wait := T#1000ms;

                IF #lfb_TON_Wait.Q THEN
                    #lx_Start_TON_Wait := FALSE;
                    #li_StepCase := 120;
                END_IF;

            120:    // парковка вертикальной оси
                "gtyp_VGR".vertical_Axis.x_Reference := TRUE;
                IF NOT "gtyp_VGR".vertical_Axis.x_Referenced THEN
                    #li_StepCase := 130;
                END_IF;

            130:    // завершение парковки вертикальной оси
                IF "gtyp_VGR".vertical_Axis.x_Referenced THEN
                    "gtyp_VGR".vertical_Axis.x_Reference := FALSE;
                    #li_StepCase := 140;
                END_IF;

           (***********************************************************)
           (****  Переместить деталь на механизм загрузки в печь,  ****)
           (****  затем захватить деталь с механизма загрузки      ****)
           (***********************************************************)

           140:  // вращение платформы
               "gtyp_VGR".rotate_Axis.di_Target_Position := "gtyp_VGR".di_Pos_MPO_rotate;
                "gtyp_VGR".rotate_Axis.x_Start_Positioning := TRUE;

                IF ("gtyp_VGR".rotate_Axis.di_Actual_Position <= ("gtyp_VGR".di_Pos_MPO_rotate + "gtyp_VGR".rotate_Axis.Config.di_Pos_Window))
                    AND ("gtyp_VGR".rotate_Axis.di_Actual_Position >= ("gtyp_VGR".di_Pos_MPO_rotate - "gtyp_VGR".rotate_Axis.Config.di_Pos_Window))
                    AND "gtyp_VGR".rotate_Axis.x_Position_Reached THEN
                    "gtyp_VGR".rotate_Axis.x_Start_Positioning := FALSE;
                    #li_StepCase := 150;
                END_IF;

            150:   // горизонтальная ось вперед
                "gtyp_VGR".horizontal_Axis.di_Target_Position := "gtyp_VGR".di_Pos_MPO_horizontal;
                "gtyp_VGR".horizontal_Axis.x_Start_Positioning := TRUE;

                IF ("gtyp_VGR".horizontal_Axis.di_Actual_Position <= ("gtyp_VGR".di_Pos_MPO_horizontal + "gtyp_VGR".horizontal_Axis.Config.di_Pos_Window))
                    AND ("gtyp_VGR".horizontal_Axis.di_Actual_Position >= ("gtyp_VGR".di_Pos_MPO_horizontal - "gtyp_VGR".horizontal_Axis.Config.di_Pos_Window))
                    AND "gtyp_VGR".horizontal_Axis.x_Position_Reached THEN
                    "gtyp_VGR".horizontal_Axis.x_Start_Positioning := FALSE;
                    #li_StepCase := 160;
                END_IF;

            160:   // вертикальная ось вниз
                "gtyp_VGR".vertical_Axis.di_Target_Position := "gtyp_VGR".di_Pos_MPO_vertical;
                "gtyp_VGR".vertical_Axis.x_Start_Positioning := TRUE;

                IF ("gtyp_VGR".vertical_Axis.di_Actual_Position <= ("gtyp_VGR".di_Pos_MPO_vertical + "gtyp_VGR".vertical_Axis.Config.di_Pos_Window))
                    AND ("gtyp_VGR".vertical_Axis.di_Actual_Position >= ("gtyp_VGR".di_Pos_MPO_vertical - "gtyp_VGR".vertical_Axis.Config.di_Pos_Window))
                    AND "gtyp_VGR".vertical_Axis.x_Position_Reached THEN
                    "gtyp_VGR".vertical_Axis.x_Start_Positioning := FALSE;
                    #li_StepCase := 170;
                END_IF;

            170:   // выключение клапана и компрессора (отпустить деталь)
                "QX_VGR_ValveVacuum_Q8" := FALSE;
                "QX_VGR_Compressor_Q7" := FALSE;

                #lx_Start_TON_Wait := TRUE;
                #lt_TON_Wait := T#500ms;
                IF #lfb_TON_Wait.Q THEN
                    #lx_Start_TON_Wait := FALSE;
                    #li_StepCase := 180;
                END_IF;

            180:   // вертикальная ось вверх
                "gtyp_VGR".vertical_Axis.di_Target_Position := "gtyp_VGR".di_Pos_MPO_vertical - "gtyp_VGR".di_Offset_Pos_MPO_vertical;
                "gtyp_VGR".vertical_Axis.x_Start_Positioning := TRUE;

                IF ("gtyp_VGR".vertical_Axis.di_Actual_Position <= ("gtyp_VGR".di_Pos_MPO_vertical - "gtyp_VGR".di_Offset_Pos_MPO_vertical + "gtyp_VGR".vertical_Axis.Config.di_Pos_Window))
                    AND ("gtyp_VGR".vertical_Axis.di_Actual_Position >= ("gtyp_VGR".di_Pos_MPO_vertical - "gtyp_VGR".di_Offset_Pos_MPO_vertical - "gtyp_VGR".vertical_Axis.Config.di_Pos_Window))
                    AND "gtyp_VGR".vertical_Axis.x_Position_Reached THEN
                    "gtyp_VGR".vertical_Axis.x_Start_Positioning := FALSE;
                    #li_StepCase := 200;
                END_IF;


           200:   // вертикальная ось вниз
                "gtyp_VGR".vertical_Axis.di_Target_Position := "gtyp_VGR".di_Pos_MPO_vertical;
                "gtyp_VGR".vertical_Axis.x_Start_Positioning := TRUE;

                IF ("gtyp_VGR".vertical_Axis.di_Actual_Position <= ("gtyp_VGR".di_Pos_MPO_vertical + "gtyp_VGR".vertical_Axis.Config.di_Pos_Window))
                    AND ("gtyp_VGR".vertical_Axis.di_Actual_Position >= ("gtyp_VGR".di_Pos_MPO_vertical - "gtyp_VGR".vertical_Axis.Config.di_Pos_Window))
                    AND "gtyp_VGR".vertical_Axis.x_Position_Reached THEN
                    "gtyp_VGR".vertical_Axis.x_Start_Positioning := FALSE;
                    #li_StepCase := 210;
                END_IF;

            210:   // запуск компрессора
                "QX_VGR_Compressor_Q7" := TRUE;

                #lx_Start_TON_Wait := TRUE;
                #lt_TON_Wait := T#1000ms;

                IF #lfb_TON_Wait.Q THEN
                    #lx_Start_TON_Wait := FALSE;
                    #li_StepCase := 220;
                END_IF;

           220:   // включение клапана (захват детали)
                "QX_VGR_ValveVacuum_Q8" := true;

                #lx_Start_TON_Wait := TRUE;
                #lt_TON_Wait := T#1000ms;

                IF #lfb_TON_Wait.Q THEN
                    #lx_Start_TON_Wait := FALSE;
                    #li_StepCase := 230;
                END_IF;

            230:   // парковка вертикальной оси
                "gtyp_VGR".vertical_Axis.x_Reference := TRUE;
                IF NOT "gtyp_VGR".vertical_Axis.x_Referenced THEN
                    #li_StepCase := 240;
                END_IF;

            240:   // завершение парковки вертикальной оси
                IF "gtyp_VGR".vertical_Axis.x_Referenced THEN
                    "gtyp_VGR".vertical_Axis.x_Reference := FALSE;
                    #li_StepCase := 250;
                END_IF;

            250:   // парковка горизонтальной оси
                "gtyp_VGR".horizontal_Axis.x_Reference := TRUE;

                IF NOT "gtyp_VGR".horizontal_Axis.x_Referenced THEN
                    #li_StepCase := 260;
                END_IF;

            260:   // завершение парковки горизонтальной оси
                IF "gtyp_VGR".horizontal_Axis.x_Referenced THEN
                    "gtyp_VGR".horizontal_Axis.x_Reference := FALSE;
                    #li_StepCase := 270;
                END_IF;

            (*************************************************************************)
            (****  Поместить деталь в карман белых деталей, затем повторить цикл  ****)
            (*************************************************************************)

            270:   // вращение платформы
                "gtyp_VGR".rotate_Axis.di_Target_Position := "gtyp_VGR".di_Pos_SLD_White_rotate;
                "gtyp_VGR".rotate_Axis.x_Start_Positioning := TRUE;

                IF ("gtyp_VGR".rotate_Axis.di_Actual_Position <= ("gtyp_VGR".di_Pos_SLD_White_rotate + "gtyp_VGR".rotate_Axis.Config.di_Pos_Window))
                    AND ("gtyp_VGR".rotate_Axis.di_Actual_Position >= ("gtyp_VGR".di_Pos_SLD_White_rotate - "gtyp_VGR".rotate_Axis.Config.di_Pos_Window))
                    AND "gtyp_VGR".rotate_Axis.x_Position_Reached THEN
                    "gtyp_VGR".rotate_Axis.x_Start_Positioning := FALSE;
                    #li_StepCase := 280;
                END_IF;

            280:   // горизонтальная ось вперед
                "gtyp_VGR".horizontal_Axis.di_Target_Position := "gtyp_VGR".di_Pos_SLD_White_horizontal;
                "gtyp_VGR".horizontal_Axis.x_Start_Positioning := TRUE;

                IF ("gtyp_VGR".horizontal_Axis.di_Actual_Position <= ("gtyp_VGR".di_Pos_SLD_White_horizontal + "gtyp_VGR".horizontal_Axis.Config.di_Pos_Window))
                    AND ("gtyp_VGR".horizontal_Axis.di_Actual_Position >= ("gtyp_VGR".di_Pos_SLD_White_horizontal - "gtyp_VGR".horizontal_Axis.Config.di_Pos_Window))
                    AND "gtyp_VGR".horizontal_Axis.x_Position_Reached THEN
                    "gtyp_VGR".horizontal_Axis.x_Start_Positioning := FALSE;
                    #li_StepCase := 290;
                END_IF;

            290:   // вертикальная ось вниз
                "gtyp_VGR".vertical_Axis.di_Target_Position := "gtyp_VGR".di_Pos_SLD_White_vertical;
                "gtyp_VGR".vertical_Axis.x_Start_Positioning := TRUE;

                IF ("gtyp_VGR".vertical_Axis.di_Actual_Position <= ("gtyp_VGR".di_Pos_SLD_White_vertical + "gtyp_VGR".vertical_Axis.Config.di_Pos_Window))
                    AND ("gtyp_VGR".vertical_Axis.di_Actual_Position >= ("gtyp_VGR".di_Pos_SLD_White_vertical - "gtyp_VGR".vertical_Axis.Config.di_Pos_Window))
                    AND "gtyp_VGR".vertical_Axis.x_Position_Reached THEN
                    "gtyp_VGR".vertical_Axis.x_Start_Positioning := FALSE;
                    #li_StepCase := 300;
                END_IF;

            300:   // выключение клапана
                "QX_VGR_ValveVacuum_Q8" := FALSE;
                #lx_Start_TON_Wait := TRUE;
                #lt_TON_Wait := T#500ms;
                IF #lfb_TON_Wait.Q THEN
                    #lx_Start_TON_Wait := FALSE;
                    #li_StepCase := 10;
                END_IF;
       END_CASE;
   END_IF;
END_FUNCTION_BLOCK

FUNCTION_BLOCK "PRG_VGR_Axis_horizontal"   // FB4, SCL
TITLE = Program Axis horizontal VGR
{ S7_Optimized_Access := 'TRUE' }
AUTHOR : A.Schaefer
VERSION : 0.0
   VAR
      lx_Init : Bool;
      lfb_horizontal_Axis : "FB_Axis";
   END_VAR
BEGIN
   IF #lx_Init THEN

       // FB Axis horizontal
       #lfb_horizontal_Axis(ini_Axis       := 1,
                   indi_Increment          := "gtyp_VGR".horizontal_Axis.di_Increment,
                   inx_Ref_Switch          := "IX_VGR_RefSwitchHorizontalAxis_I2",
                   inx_Referencing         := "gtyp_VGR".horizontal_Axis.x_Reference,
                   inx_Start_Positioning   := "gtyp_VGR".horizontal_Axis.x_Start_Positioning,
                   indi_Target_Position    := "gtyp_VGR".horizontal_Axis.di_Target_Position,
                   ini_PWM                 := "gtyp_VGR".horizontal_Axis.i_PWM,
                   inouttyp_Config         := "gtyp_VGR".horizontal_Axis.Config,
                   inouttyp_Setup          := "gtyp_SetupAxis");

       "QX_VGR_M2_HorizontalAxisForward_Q4"    := #lfb_horizontal_Axis.outx_Motor_Pos;
       "QX_VGR_M2_HorizontalAxisBackward_Q3"   := #lfb_horizontal_Axis.outx_Motor_Neg;
       "gtyp_VGR".horizontal_Axis.di_Actual_Position    := #lfb_horizontal_Axis.outdi_Actual_Position;
       "gtyp_VGR".horizontal_Axis.x_Referenced          := #lfb_horizontal_Axis.outx_Referenced;
       "gtyp_VGR".horizontal_Axis.x_Position_Reached    := #lfb_horizontal_Axis.outx_Position_Reached;
   ELSE
       #lx_Init := TRUE;
   END_IF;
END_FUNCTION_BLOCK

FUNCTION_BLOCK "PRG_VGR_Axis_rotate"   // FB5, SCL
TITLE = Program Axis rotate VGR
{ S7_Optimized_Access := 'TRUE' }
AUTHOR : A.Schaefer
VERSION : 0.0
   VAR
      lx_Init : Bool;
      lfb_rotate_Axis : "FB_Axis";
   END_VAR
BEGIN
   IF #lx_Init THEN

       // FB Axis rotate
       #lfb_rotate_Axis(ini_Axis           := 3,
                   indi_Increment          := "gtyp_VGR".rotate_Axis.di_Increment,
                   inx_Ref_Switch          := "IX_VGR_RefSwitchRotate_I3",
                   inx_Referencing         := "gtyp_VGR".rotate_Axis.x_Reference,
                   inx_Start_Positioning   := "gtyp_VGR".rotate_Axis.x_Start_Positioning,
                   indi_Target_Position    := "gtyp_VGR".rotate_Axis.di_Target_Position,
                   ini_PWM                 := "gtyp_VGR".rotate_Axis.i_PWM,
                   inouttyp_Config         := "gtyp_VGR".rotate_Axis.Config,
                   inouttyp_Setup          := "gtyp_SetupAxis");

       "QX_VGR_M3_RotateClockwise_Q5"          := #lfb_rotate_Axis.outx_Motor_Neg;
       "QX_VGR_M3_RotateCounterclockwise_Q6"   := #lfb_rotate_Axis.outx_Motor_Pos;
       "gtyp_VGR".rotate_Axis.di_Actual_Position := #lfb_rotate_Axis.outdi_Actual_Position;
       "gtyp_VGR".rotate_Axis.x_Referenced       := #lfb_rotate_Axis.outx_Referenced;
       "gtyp_VGR".rotate_Axis.x_Position_Reached := #lfb_rotate_Axis.outx_Position_Reached;
   ELSE
       #lx_Init := TRUE;
   END_IF;
END_FUNCTION_BLOCK

FUNCTION_BLOCK "PRG_VGR_Axis_vertical_Act_Pos"   // FB28, SCL
TITLE = Program Axis vertical Actual Position VGR
{ S7_Optimized_Access := 'TRUE' }
AUTHOR : A.Schaefer
VERSION : 0.0
   VAR
      lfb_IN_DEC : "FB_INC_DEC";
      lfb_Axis : "FB_Axis";
   END_VAR
BEGIN
   "CTRL_HSC_0_DB"(HSC:="Local~HSC_3",
                   CV:="IX_VGR_RefSwitchVerticalAxis_I1",
                   NEW_CV:= 0);

   "gtyp_VGR".vertical_Axis.di_Increment := "Enc_VGR_vertical";
END_FUNCTION_BLOCK

FUNCTION_BLOCK "PRG_VGR_Axis_horizontal_Act_Pos"   // FB29, SCL
TITLE = Program Axis horizontal Actual Position VGR
{ S7_Optimized_Access := 'TRUE' }
AUTHOR : A.Schaefer
VERSION : 0.0
   VAR
      lfb_IN_DEC : "FB_INC_DEC";
      lfb_Axis : "FB_Axis";
   END_VAR
BEGIN
   "CTRL_HSC_1_DB"(HSC:="Local~HSC_4",
                   CV:="IX_VGR_RefSwitchHorizontalAxis_I2",
                   NEW_CV:= 0);

   "gtyp_VGR".horizontal_Axis.di_Increment := "Enc_VGR_horizontal";
END_FUNCTION_BLOCK

FUNCTION_BLOCK "PRG_VGR_Axis_rotate_Act_Pos"   // FB30, SCL
TITLE = Program Axis rotate Actual Position VGR
{ S7_Optimized_Access := 'TRUE' }
AUTHOR : A.Schaefer
VERSION : 0.0
   VAR
      lfb_IN_DEC : "FB_INC_DEC";
      lfb_Axis : "FB_Axis";
   END_VAR
BEGIN
   "CTRL_HSC_2_DB"(HSC:="Local~HSC_5",
                   CV:="IX_VGR_RefSwitchRotate_I3",
                   NEW_CV:= 0);

   "gtyp_VGR".rotate_Axis.di_Increment := "Enc_VGR_rotate";
END_FUNCTION_BLOCK